// Mitsubishi GX Works2 project: BookEX3_5 Data   PLC: Q13UDV

TYPE DateTime : STRUCT
  Year : INT;
  Month : INT;
  Day : INT;
  WeekDay : INT;
  iHour : INT;
  iMin : INT;
  iSec : INT;
  ms : INT;
END_STRUCT END_TYPE

TYPE Vector : STRUCT
  axisX : REAL;
  axisY : REAL;
  axisZ : REAL;
END_STRUCT END_TYPE

TYPE WordBit : STRUCT
  Data : DWORD;
  Flag : BOOL;
END_STRUCT END_TYPE

// global labels: Global
VAR_GLOBAL
  bVar0 AT M5000 : BOOL;
  abArray0 AT M5010 : ARRAY [0..49] OF BOOL;
  sStr0 AT D5000 : STRING[199];
  sStr1 AT D5100 : STRING[199];
  sStr2 AT D5200 : STRING[199];
  sStr3 AT D5300 : STRING[199];
  sStr4 AT D5400 : STRING[199];
  sStr5 AT D5500 : STRING[199];
  sStr6 AT D5600 : STRING[199];
  sStr7 AT D5700 : STRING[199];
  sStr8 AT D5800 : STRING[199];
  sStr9 AT D5900 : STRING[199];
  iVar0 AT D4500 : INT;
  iVar1 AT D4501 : INT;
  iVar2 AT D4502 : INT;
  iVar3 AT D4503 : INT;
  iVar4 AT D4504 : INT;
  iVar5 AT D4505 : INT;
  iVar6 AT D4506 : INT;
  iVar7 AT D4507 : INT;
  iVar8 AT D4508 : INT;
  iVar9 AT D4509 : INT;
  dVar0 AT D4510 : DINT;
  dVar1 AT D4512 : DINT;
  dVar2 AT D4514 : DINT;
  dVar3 AT D4516 : DINT;
  dVar4 AT D4518 : DINT;
  dVar5 AT D4520 : DINT;
  dVar6 AT D4522 : DINT;
  dVar7 AT D4524 : DINT;
  dVar8 AT D4526 : DINT;
  dVar9 AT D4528 : DINT;
  wVar0 AT D4530 : WORD;
  wVar1 AT D4531 : WORD;
  wVar2 AT D4532 : WORD;
  wVar3 AT D4533 : WORD;
  wVar4 AT D4534 : WORD;
  wVar5 AT D4535 : WORD;
  wVar6 AT D4536 : WORD;
  wVar7 AT D4537 : WORD;
  wVar8 AT D4538 : WORD;
  wVar9 AT D4539 : WORD;
  dwVar0 AT D4540 : DWORD;
  dwVar1 AT D4542 : DWORD;
  dwVar2 AT D4544 : DWORD;
  dwVar3 AT D4546 : DWORD;
  dwVar4 AT D4548 : DWORD;
  dwVar5 AT D4550 : DWORD;
  dwVar6 AT D4552 : DWORD;
  dwVar7 AT D4554 : DWORD;
  dwVar8 AT D4556 : DWORD;
  dwVar9 AT D4558 : DWORD;
  fsVar0 AT D4560 : REAL;
  fsVar1 AT D4562 : REAL;
  fsVar2 AT D4564 : REAL;
  fsVar3 AT D4566 : REAL;
  fsVar4 AT D4568 : REAL;
  fsVar5 AT D4570 : REAL;
  fsVar6 AT D4572 : REAL;
  fsVar7 AT D4574 : REAL;
  fsVar8 AT D4576 : REAL;
  fsVar9 AT D4578 : REAL;
  fdVar0 AT D4580 : LREAL;
  tTime0 AT D4620 : TIME;
  tTime1 AT D4622 : TIME;
  tTime2 AT D4624 : TIME;
  tTime3 AT D4626 : TIME;
  tTime4 AT D4628 : TIME;
  tTime5 AT D4630 : TIME;
  tTime6 AT D4632 : TIME;
  tTime7 AT D4634 : TIME;
  tTime8 AT D4636 : TIME;
  tTime9 AT D4638 : TIME;
  tTime10 AT D4640 : TIME;
  bVar1 AT M5001 : BOOL;
  bVar2 AT M5002 : BOOL;
  bVar3 AT M5003 : BOOL;
  bVar4 AT M5004 : BOOL;
  bVar5 AT M5005 : BOOL;
  bVar6 AT M5006 : BOOL;
  bVar7 AT M5007 : BOOL;
  bVar8 AT M5008 : BOOL;
  bVar9 AT M5009 : BOOL;
  abArray1 AT M5060 : ARRAY [0..49] OF BOOL;
  abArray2 AT M5110 : ARRAY [0..49] OF BOOL;
  abArray3 AT M5160 : ARRAY [0..49] OF BOOL;
  abArray4 AT M5210 : ARRAY [0..49] OF BOOL;
  abArray5 AT M5260 : ARRAY [0..49] OF BOOL;
  abArray6 AT M5310 : ARRAY [0..49] OF BOOL;
  abArray7 AT M5360 : ARRAY [0..49] OF BOOL;
  abArray8 AT M5410 : ARRAY [0..49] OF BOOL;
  abArray9 AT M5460 : ARRAY [0..49] OF BOOL;
  fdVar1 AT D4584 : LREAL;
  fdVar2 AT D4588 : LREAL;
  fdVar3 AT D4592 : LREAL;
  fdVar4 AT D4596 : LREAL;
  fdVar5 AT D4600 : LREAL;
  fdVar6 AT D4604 : LREAL;
  fdVar7 AT D4608 : LREAL;
  fdVar8 AT D4612 : LREAL;
  fdVar9 AT D4616 : LREAL;
  aSendData1 AT D100 : ARRAY [0..9] OF INT;
  aiTxData AT D4000 : ARRAY [0..99] OF INT;
  aiRxData AT D4100 : ARRAY [0..99] OF INT;
  iOpenOK AT D3900 : INT;
  iOpenERR AT D3901 : INT;
  iSendOK AT D3902 : INT;
  iSendERR AT D3903 : INT;
  iCloseOK AT D3906 : INT;
  iCloseERR AT D3907 : INT;
  iRecvOK AT D3904 : INT;
  iRecvERR AT D3905 : INT;
  aiTxData2 AT D4200 : ARRAY [0..99] OF INT;
  aiRxData2 AT D4300 : ARRAY [0..99] OF INT;
  iOpenOK2 AT D3908 : INT;
  iOpenERR2 AT D3909 : INT;
  iSendOK2 AT D3910 : INT;
  iSendERR2 AT D3911 : INT;
  iRecvOK2 AT D3912 : INT;
  iRecvERR2 AT D3913 : INT;
  iCloseOK2 AT D3914 : INT;
  iCloseERR2 AT D3915 : INT;
  iEOpenComp AT D3916 : INT;
  iEOpenReq AT D3917 : INT;
  iERecvFlag AT D3918 : INT;
  iOpenCode AT D3919 : INT;
  iSendCode AT D3920 : INT;
  iRecvCode AT D3921 : INT;
  iCloseCode AT D3922 : INT;
  iOpenCode2 AT D3923 : INT;
  iSendCode2 AT D3924 : INT;
  iRecvCode2 AT D3925 : INT;
  iCloseCode2 AT D3926 : INT;
  aRecvData1 AT D110 : ARRAY [0..9] OF INT;
  aSendData2 AT D120 : ARRAY [0..9] OF INT;
  aRecvData2 AT D130 : ARRAY [0..9] OF INT;
END_VAR
// user libraries (not included): HMI

FUNCTION_BLOCK AllFB
VAR_INPUT
  b_IN1 : BOOL;
  b_IN2 : BOOL;
END_VAR
VAR_OUTPUT
  b_OT : BOOL;
END_VAR
(* structured ladder/FBD written out as ST: instructions are called as NAME(EN, inputs, outputs); _pN, _eN, _tN stand for wires *)
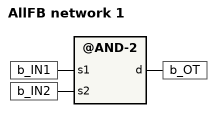
(* network 1 *)
b_OT := @AND-2(b_IN1, b_IN2);
END_FUNCTION_BLOCK

FUNCTION_BLOCK EnFB
VAR_INPUT
  b_IN1 : BOOL;
  b_IN2 : BOOL;
END_VAR
VAR_OUTPUT
  b_OT : BOOL;
END_VAR
(* structured ladder/FBD written out as ST: instructions are called as NAME(EN, inputs, outputs); _pN, _eN, _tN stand for wires *)
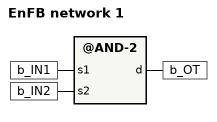
(* network 1 *)
b_OT := @AND-2(b_IN1, b_IN2);
END_FUNCTION_BLOCK

FUNCTION EnFUN
VAR_INPUT
  b_IN1 : BOOL;
  b_IN2 : BOOL;
END_VAR
(* structured ladder/FBD written out as ST: instructions are called as NAME(EN, inputs, outputs); _pN, _eN, _tN stand for wires *)
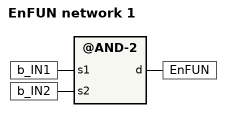
(* network 1 *)
EnFUN := @AND-2(b_IN1, b_IN2);
END_FUNCTION

FUNCTION_BLOCK MacroEnFB
VAR_INPUT
  b_IN1 : BOOL;
  b_IN2 : BOOL;
END_VAR
VAR_OUTPUT
  b_OT : BOOL;
END_VAR
(* structured ladder/FBD written out as ST: instructions are called as NAME(EN, inputs, outputs); _pN, _eN, _tN stand for wires *)
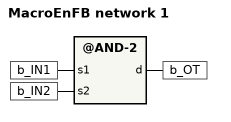
(* network 1 *)
b_OT := @AND-2(b_IN1, b_IN2);
END_FUNCTION_BLOCK

FUNCTION_BLOCK MacroFB
VAR_INPUT
  b_IN1 : BOOL;
  b_IN2 : BOOL;
END_VAR
VAR_OUTPUT
  b_OT : BOOL;
END_VAR
VAR
  ix : INT;
END_VAR
(* structured ladder/FBD written out as ST: instructions are called as NAME(EN, inputs, outputs); _pN, _eN, _tN stand for wires *)
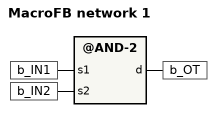
(* network 1 *)
b_OT := @AND-2(b_IN1, b_IN2);
END_FUNCTION_BLOCK

FUNCTION_BLOCK ManEnFB
VAR_INPUT
  b_EN : BOOL;
  b_IN2 : BOOL;
END_VAR
VAR_OUTPUT
  b_OT : BOOL;
END_VAR
VAR
  ix : INT;
END_VAR
VAR_INPUT
  b_IN1 : BOOL;
END_VAR
VAR_OUTPUT
  b_ENO : BOOL;
END_VAR
(* structured ladder/FBD written out as ST: instructions are called as NAME(EN, inputs, outputs); _pN, _eN, _tN stand for wires *)
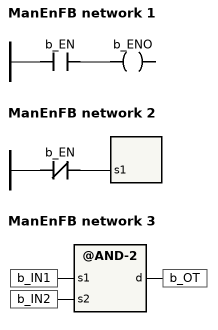
(* network 1 *)
b_ENO := b_EN;
(* network 2 *)
(* element kind 10  <- NOT b_EN *)
(* network 3 *)
b_OT := @AND-2(b_IN1, b_IN2);
END_FUNCTION_BLOCK

FUNCTION_BLOCK NoneFB
VAR_INPUT
  b_IN1 : BOOL;
  b_IN2 : BOOL;
END_VAR
VAR_OUTPUT
  b_OT : BOOL;
END_VAR
(* structured ladder/FBD written out as ST: instructions are called as NAME(EN, inputs, outputs); _pN, _eN, _tN stand for wires *)
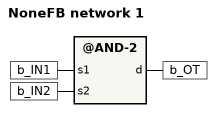
(* network 1 *)
b_OT := @AND-2(b_IN1, b_IN2);
END_FUNCTION_BLOCK

FUNCTION NoneFUN
VAR_INPUT
  b_IN1 : BOOL;
  b_IN2 : BOOL;
END_VAR
(* structured ladder/FBD written out as ST: instructions are called as NAME(EN, inputs, outputs); _pN, _eN, _tN stand for wires *)
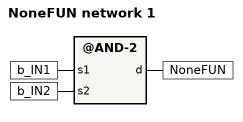
(* network 1 *)
NoneFUN := @AND-2(b_IN1, b_IN2);
END_FUNCTION

FUNCTION_BLOCK ScanInput
VAR_INPUT
  Inp : BOOL;
END_VAR
VAR_OUTPUT
  UpEg : BOOL;
END_VAR
VAR
  CurrBit : BOOL;
  LastBit : BOOL;
END_VAR
VAR_OUTPUT
  DwEg : BOOL;
  Last : BOOL;
END_VAR
;
CurrBit := Inp;
UpEg := CurrBit AND NOT LastBit;
DwEg := NOT CurrBit AND LastBit;
Last := LastBit;
LastBit := CurrBit;
END_FUNCTION_BLOCK

FUNCTION_BLOCK wireTXD
VAR_INPUT
  CurX : INT;
  wFork : WORD;
  wKind : INT;
  LedF2 : WORD;
  LedF1 : WORD;
  CurY : INT;
END_VAR
VAR_OUTPUT
  DPhs : INT;
  TxBit3 : BOOL;
  TxBit2 : BOOL;
  TxBit1 : BOOL;
  TxBit0 : BOOL;
  TxClock : BOOL;
END_VAR
VAR
  Phase : INT;
  MaskBit : WORD;
END_VAR
VAR_OUTPUT
  Dmask : WORD;
END_VAR
VAR
  TD3 : WORD;
  TD2 : WORD;
  TD1 : WORD;
  TD0 : WORD;
END_VAR
VAR_INPUT
  wBank : WORD;
  wX : INT;
  wY : INT;
  ErrC : INT;
  MacNo : INT;
END_VAR
VAR
  ix : INT;
END_VAR
VAR_INPUT
  Debug1 : WORD;
  Debug2 : WORD;
  Debug : BOOL;
  Boot : BOOL;
  BootSts : WORD;
  BootTime : DINT;
END_VAR
VAR
  SaveTD0 : WORD;
  SaveTD1 : WORD;
  wTmp : WORD;
END_VAR
VAR_OUTPUT
  TxData0 : WORD;
  TxData1 : WORD;
  TxData2 : WORD;
  TxData3 : WORD;
END_VAR
VAR
  iy : INT;
END_VAR
;

IF Phase = 0 OR Phase > 35 THEN
	(* Data준비 *)	
	IF gbModeManual THEN
		TD0 := 16#0000;	
		IF orBox[0] THEN TD0 := TD0 OR 16#0100; END_IF;
		IF orBox[1] THEN TD0 := TD0 OR 16#0200; END_IF;
		IF orBox[2] THEN TD0 := TD0 OR 16#0400; END_IF;
		IF orBox[3] THEN TD0 := TD0 OR 16#0800; END_IF;
		TD1 := INT_TO_WORD(CurX * 256 + CurY);
		TD0 := TD0 OR INT_TO_WORD(MacNo);
   		TD2 := LedF1; 
   		TD3 := LedF2; 
	ELSE
		TD0 := wFork;
		TD0 := SHL(TD0, 8) AND 16#FF00;
		TD0 := TD0 OR 16#0080;	
	END_IF;
	IF gbAlarm THEN 
		TD0 := TD0 OR 16#0040;
		TD1 := INT_TO_WORD(ErrC); 
   		TD2 := LedF1;  
   		TD3 := LedF2; 
	ELSIF Debug  THEN	
 		TD0 := Debug1;
 		TD1 := Debug2;
   		TD2 := LedF1 OR 16#2000; 
   		TD3 := LedF2; 
	ELSIF Boot THEN
		TD0 := TD0 OR 16#0020 OR INT_TO_WORD(MacNo);
 		TD1 := DINT_TO_WORD(BootTime/1000);
   		TD2 := BootSts; 
		TD3 := BootSts;   		
	 ELSIF NOT gbModeManual  THEN
		wTmp := SHL(INT_TO_WORD( jobDispKind ) AND 16#000F, 12); 	
		iy := Bank_TO_INT(wBank);
			IF MacNo > 5 THEN
				ix := MacNo*4-iy+1;
			ELSE
				ix := MacNo*4+iy-4;
			END_IF;
			
   		CASE jobDispKind  OF
   			0 :  
					TD0 := TD0 OR wTmp;	
 					TD1 := 0;
			1,2 :  
					TD0 := TD0 OR wTmp;	
 					TD1 := 1;
			3,4 :  
					TD0 := TD0 OR wTmp;	
 					TD1 := 2;
   			5,11,12 : 
					TD0 := TD0 OR wTmp;	
 					TD1 := INT_TO_WORD(jobDispKind)  ;
			6,7,8 :  			
					TD0 := TD0 OR wTmp OR INT_TO_WORD(ix);;	
 					TD1 := INT_TO_WORD(wX * 256 + wY);
			9,10 :  					
					TD0 := TD0 OR wTmp OR INT_TO_WORD(ix);;	
 					TD1 := INT_TO_WORD(wX * 256 + wY);
			13,14,15 :  
					TD0 := TD0 OR wTmp;	
					TD1 := wFork;
		ELSE
			TD0 := 16#0080;	
 			TD1 := 0;
		END_CASE;	
   		TD2 := LedF1;  
   		TD3 := LedF2; 
	END_IF;
 		
		TxClock := TRUE;
		TxBit0 := TRUE;	
		TxBit1 := TRUE;	
		TxBit2 := TRUE;	
		TxBit3 := TRUE;	
		Phase := 1;
ELSIF Phase = 1 THEN
     (* ON Start Bit F *)	
    	TxClock := FALSE;
		TxBit0 := TRUE;	
		TxBit1 := TRUE;	
		TxBit2 := TRUE;	
		TxBit3 := TRUE;	
		Phase := 2;
		MaskBit := 16#8000;
ELSIF Phase = 34 THEN
    (* ON Stop *)	
    	TxClock := TRUE;
		TxBit0 := FALSE;	
		TxBit1 := FALSE;	
		TxBit2 := FALSE;	
		TxBit3 := FALSE;	
		Phase := 35;
ELSIF Phase = 35 THEN
     (* OFF Stop *)	
    	TxClock := FALSE;
		TxBit0 := FALSE;	
		TxBit1 := FALSE;	
		TxBit2 := FALSE;	
		TxBit3 := FALSE;
		Phase := 0;	
ELSE	
		IF (MaskBit AND TD0) <> 0 THEN TxBit0 := TRUE; ELSE TxBit0 := FALSE; END_IF;
		IF (MaskBit AND TD1) <> 0 THEN TxBit1 := TRUE; ELSE TxBit1 := FALSE; END_IF;
		IF (MaskBit AND TD2) <> 0 THEN TxBit2 := TRUE; ELSE TxBit2 := FALSE; END_IF;
		IF (MaskBit AND TD3) <> 0 THEN TxBit3 := TRUE; ELSE TxBit3 := FALSE; END_IF;
	IF (Phase MOD 2) = 0 THEN
    	TxClock := TRUE;
	ELSE 
		TxClock := FALSE;
    	SFR(TRUE,1,MaskBit);
	END_IF;
	Phase := Phase + 1;
END_IF;

DPhs := Phase;
Dmask := MaskBit;
TxData0 := TD0;
TxData1 := TD1;
TxData2 := TD2;
TxData3 := TD3;
END_FUNCTION_BLOCK

PROGRAM ExComment
VAR
  HMI05_1 : HMI05;
END_VAR
(* structured ladder/FBD written out as ST: instructions are called as NAME(EN, inputs, outputs); _pN, _eN, _tN stand for wires *)
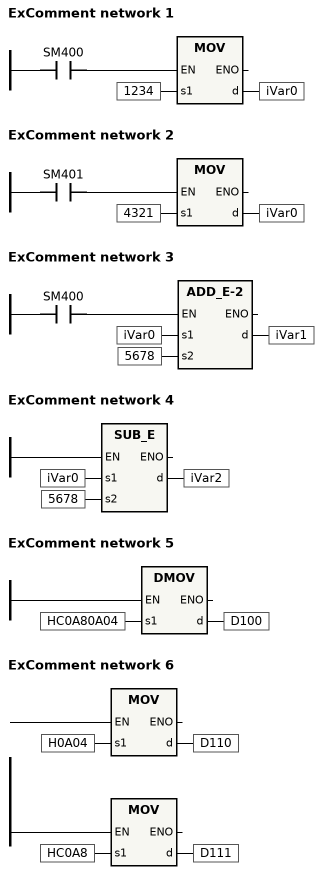
(* network 1 *)
MOV(SM400, 1234, iVar0);
(* network 2 *)
MOV(SM401, 4321, iVar0);
(* network 3 *)
ADD_E(SM400, iVar0, 5678, iVar1);
(* network 4 *)
SUB_E(TRUE, iVar0, 5678, iVar2);
(* network 5 *)
DMOV(TRUE, HC0A80A04, D100);
(* network 6 *)
MOV(TRUE, H0A04, D110);
MOV(TRUE, HC0A8, D111);
END_PROGRAM

PROGRAM ExFB
VAR
  NoneFB_1 : NoneFB;
  EnFB_1 : EnFB;
  MacroFB_1 : MacroFB;
  AllFB_1 : AllFB;
  MacroEnFB_1 : MacroEnFB;
  ManEnFB_1 : ManEnFB;
END_VAR
(* structured ladder/FBD written out as ST: instructions are called as NAME(EN, inputs, outputs); _pN, _eN, _tN stand for wires *)
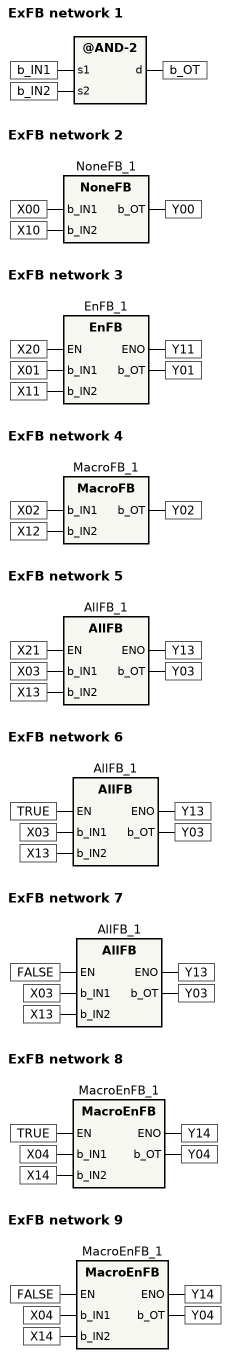
(* network 1 *)
b_OT := @AND-2(b_IN1, b_IN2);
(* network 2 *)
NoneFB_1(b_IN1 := X00, b_IN2 := X10, b_OT => Y00);
(* network 3 *)
EnFB_1(EN := X20, b_IN1 := X01, b_IN2 := X11, ENO => Y11, b_OT => Y01);
(* network 4 *)
MacroFB_1(b_IN1 := X02, b_IN2 := X12, b_OT => Y02);
(* network 5 *)
AllFB_1(EN := X21, b_IN1 := X03, b_IN2 := X13, ENO => Y13, b_OT => Y03);
(* network 6 *)
AllFB_1(EN := TRUE, b_IN1 := X03, b_IN2 := X13, ENO => Y13, b_OT => Y03);
(* network 7 *)
AllFB_1(EN := FALSE, b_IN1 := X03, b_IN2 := X13, ENO => Y13, b_OT => Y03);
(* network 8 *)
MacroEnFB_1(EN := TRUE, b_IN1 := X04, b_IN2 := X14, ENO => Y14, b_OT => Y04);
(* network 9 *)
MacroEnFB_1(EN := FALSE, b_IN1 := X04, b_IN2 := X14, ENO => Y14, b_OT => Y04);
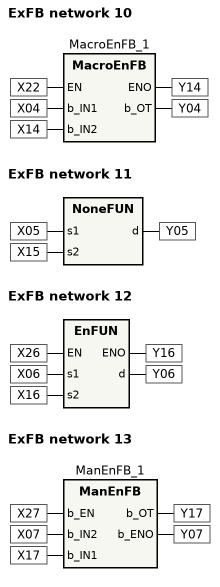
(* network 10 *)
MacroEnFB_1(EN := X22, b_IN1 := X04, b_IN2 := X14, ENO => Y14, b_OT => Y04);
(* network 11 *)
Y05 := NoneFUN(X05, X15);
(* network 12 *)
_e1 := EnFUN(X26, X06, X16, Y06);
Y16 := _e1;
(* network 13 *)
ManEnFB_1(b_EN := X27, b_IN2 := X07, b_IN1 := X17, b_OT => Y17, b_ENO => Y07);
END_PROGRAM

PROGRAM ExScanInput
VAR
  ScanInput_1 : ScanInput;
  DispHMI2_1 : DispHMI2;
END_VAR
(* structured ladder/FBD written out as ST: instructions are called as NAME(EN, inputs, outputs); _pN, _eN, _tN stand for wires *)
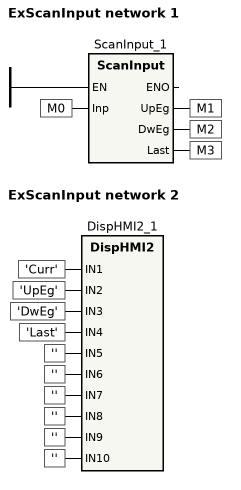
(* network 1 *)
ScanInput_1(EN := TRUE, Inp := M0, UpEg => M1, DwEg => M2, Last => M3);
(* network 2 *)
DispHMI2_1(IN1 := 'Curr', IN2 := 'UpEg', IN3 := 'DwEg', IN4 := 'Last', IN5 := '', IN6 := '', IN7 := '', IN8 := '', IN9 := '', IN10 := '');
END_PROGRAM

PROGRAM ExSHR
VAR
  Mov4WORD_1 : Mov4WORD;
  DispHMI1_1 : DispHMI1;
END_VAR
VAR CONSTANT
  cInit : INT;  (* 초기화 *)
  cStart : INT := 1;  (* 시작 *)
  cEnd : INT := 2;  (* 종료 *)
  cError : INT := 3;  (* 이상 *)
END_VAR
VAR_GLOBAL RETAIN
  iCounter : INT;
  iTarget : INT;
END_VAR
VAR
  fbLabel_1 : fbLabel;
END_VAR
(* structured ladder/FBD written out as ST: instructions are called as NAME(EN, inputs, outputs); _pN, _eN, _tN stand for wires *)
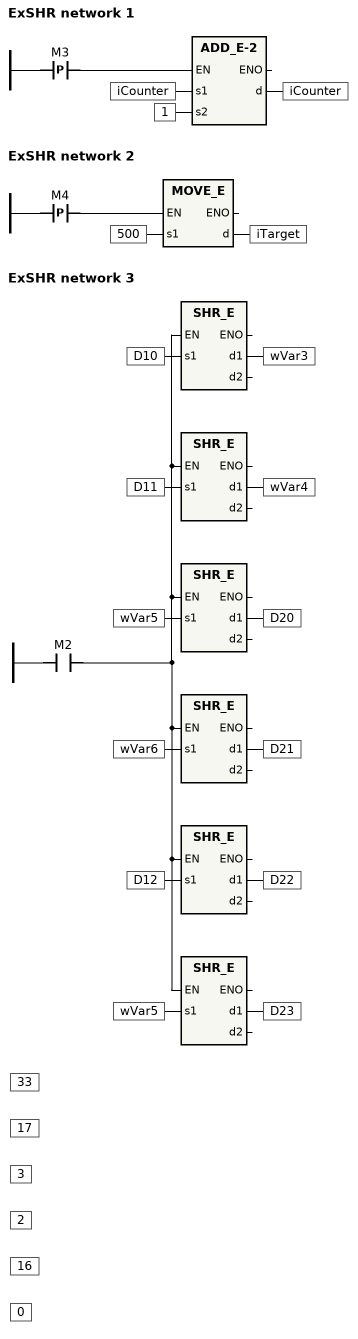
(* network 1 *)
ADD_E(LDP(TRUE, M3), iCounter, 1, iCounter);
(* network 2 *)
MOVE_E(LDP(TRUE, M4), 500, iTarget);
(* network 3 *)
SHR_E(M2, D10, wVar3, _open);
SHR_E(M2, D11, wVar4, _open);
SHR_E(M2, wVar5, D20, _open);
SHR_E(M2, wVar6, D21, _open);
SHR_E(M2, D12, D22, _open);
SHR_E(M2, wVar5, D23, _open);
(* not connected to any output: 33, 17, 3, 2, 16, 0 *)
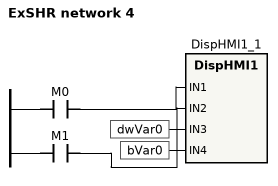
(* network 4 *)
DispHMI1_1(IN1 := M0, IN2 := M1, IN3 := dwVar0, IN4 := bVar0);
END_PROGRAM

PROGRAM ExSM701
VAR
  newBCDDA_1 : newBCDDA;
  sTemp : STRING[6];
END_VAR
(* structured ladder/FBD written out as ST: instructions are called as NAME(EN, inputs, outputs); _pN, _eN, _tN stand for wires *)
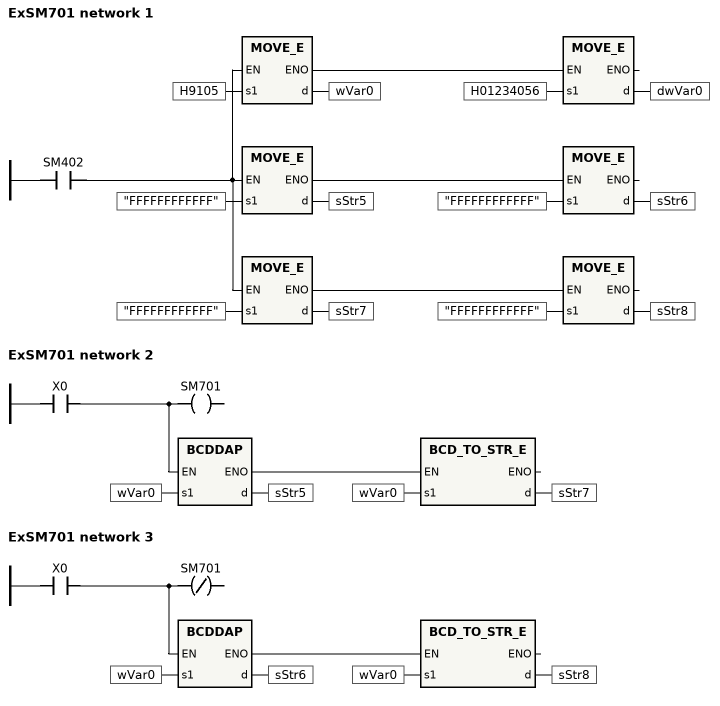
(* network 1 *)
_e1 := MOVE_E(SM402, H9105, wVar0);
MOVE_E(_e1, H01234056, dwVar0);
_e2 := MOVE_E(SM402, "FFFFFFFFFFFF", sStr5);
MOVE_E(_e2, "FFFFFFFFFFFF", sStr6);
_e3 := MOVE_E(SM402, "FFFFFFFFFFFF", sStr7);
MOVE_E(_e3, "FFFFFFFFFFFF", sStr8);
(* network 2 *)
SM701 := X0;
_e1 := BCDDAP(X0, wVar0, sStr5);
BCD_TO_STR_E(_e1, wVar0, sStr7);
(* network 3 *)
SM701 := NOT X0;
_e1 := BCDDAP(X0, wVar0, sStr6);
BCD_TO_STR_E(_e1, wVar0, sStr8);
END_PROGRAM
